// Mitsubishi GX Works2 project: 14-06-2020 LAB 2_Timer   PLC: FX3G

PROGRAM MAIN
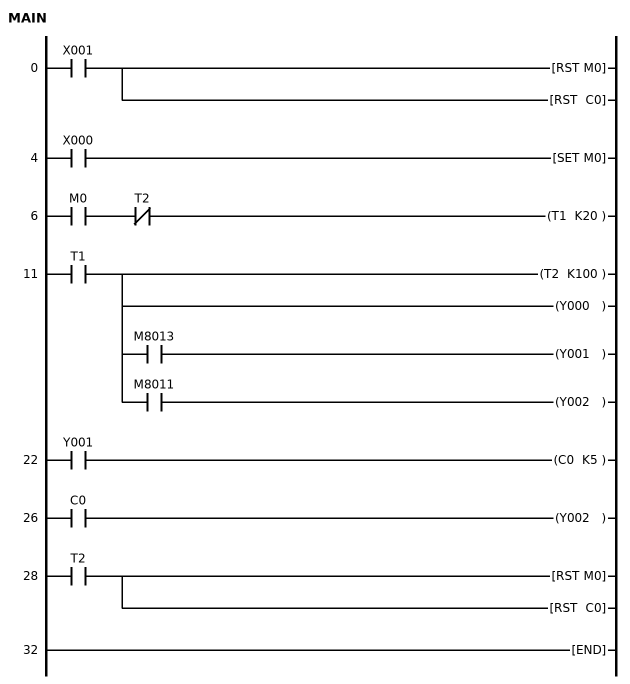
0     LD      X001
      RST     M0
      RST     C0
4     LD      X000
      SET     M0
6     LD      M0
      ANI     T2
      OUT     T1 K20
11    LD      T1
      OUT     T2 K100
      OUT     Y000
      MPS
      AND     M8013
      OUT     Y001
      MPP
      AND     M8011
      OUT     Y002
22    LD      Y001
      OUT     C0 K5
26    LD      C0
      OUT     Y002
28    LD      T2
      RST     M0
      RST     C0
32    END
END_PROGRAM
